{attribute 'GeneratedUsingTerminal: EL3773-0000-0016'}
{attribute addProperty BoxType "EL3773-0000-0016"}
{attribute addProperty Id "U3_STATUSAT %I*U3_STATUS_B07533568"}
{attribute addProperty CRC "738312571"}
{attribute addProperty Size "8"}
TYPE L3_Voltage_Status_2C01C17B EXTENDS InputBase_8311D824 :
STRUCT
	{attribute addProperty Name "U3_STATUS"}
	U3_STATUS AT %I* : U3_STATUS_B0753356;
END_STRUCT
END_TYPE

(* stored: Version 1.2.0.0, ProductVersion 3.1.4024.11
   DUT L3_Voltage_Status_2C01C17B: Id {6cd6b24b-34ad-4d47-9055-1522b449727f} *)
